# B&R Automation Studio project SampleProject
Automation Studio 4.6.7.161 SP; This is a sample project

## Configuration X20CP1586

CPU X20CP1586, AutomationRuntime B4.63, Build 4.1.2, Vc V4.62.0

### Task classes (Cpu.sw)
```
Cyclic#4:
  Program <- Program.prg
Libraries: AsNxCoM, runtime
```

### Hardware
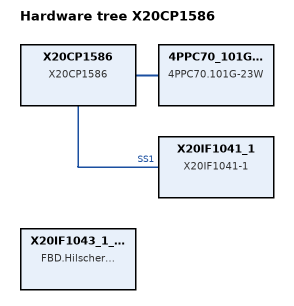
```
4PPC70_101G_23W : 4PPC70.101G-23W v1.4.0.0  [IF2 -> X20CP1586.IF2 [Cable Type=PowerlinkCable, Length=10, Version=1.0.0.2]]
  Connector IF2
  Terminal = true
  KeyMappingFile = VC\4PPC70_101G_23W1.dis
X20CP1586 : X20CP1586 v1.10.0.0
  Connector IF2:
    ActivateDevice = 1
    Mode = Manual
    InternetAddress = 10.0.0.5
    SubnetMask = 255.255.255.0
  ConfigurationID = SampleProject_X20CP1586
X20IF1041_1 : X20IF1041-1 v1.4.0.0  [SS -> X20CP1586.SS1]
  Connector IF1:
    DtmId = 2d840d1b-1473-49bf-a3aa-9ba4bb4caccd
  ConfigFile = X20IF1041_1.dtm
  ConfigModule = asnxdb1
X20IF1043_1__DTM_ : FBD.Hilscher.COGenSlaveDTM.X20IF1043-1 (BuR-X20IF1043-1.eds) v0xA70B.0x00020014 (OrderNumber=X20IF1043-1 (DTM), VendorAddress=2)
  DtmId = 
  ChannelBlocks_722b6533-4489-40d8-aae4-ca0f676f7389  // RxPDO_01
  IO_d52191ed-4c54-4aa1-a555-7a825949a8e7  // 1 Byte(s)
  IO_af2aac78-a722-4896-b9e5-1e0a5520eff8  // 1 Byte(s)
  IO_d3d611f7-76ca-4a12-9739-4a5263261990  // 1 Byte(s)
  IO_28b2f819-6018-4271-9e84-a707596ceac6  // 1 Byte(s)
  IO_602cc8aa-9b3a-44f0-8874-f1db9f83001c  // 1 Byte(s)
  IO_ddc36243-cae0-4301-b86b-f666f3c64e48  // 1 Byte(s)
  IO_1c4766d3-e1da-4921-8d87-31443da98228  // 1 Byte(s)
  IO_b8dce777-eb45-4337-9ffb-03c754224648  // 1 Byte(s)
  ChannelBlocks_8ed83e9a-ae4b-4b45-a0a9-fc1bb8b705e1  // RxPDO_02
  IO_ee120ad1-81d2-4465-b35d-721146a1a332  // 1 Byte(s)
  IO_19650846-5f72-44c2-b9fe-403733023f40  // 1 Byte(s)
  IO_7738ffe0-6403-4fb1-8263-19848970e7e6  // 1 Byte(s)
  IO_6fe8a185-5111-4af8-bbfc-95a7497bd028  // 1 Byte(s)
  IO_049ba4af-e80a-4ae3-8440-0f18dcbcee35  // 1 Byte(s)
  IO_8b1abd60-5eef-4bde-acd4-b9ff9ef701bf  // 1 Byte(s)
  IO_d0747008-f825-4f1e-bb1b-93a7cf56cb81  // 1 Byte(s)
  IO_c2f4c436-f256-4d0e-8b66-210290ce442f  // 1 Byte(s)
  ChannelBlocks_1db14d39-2e65-4f01-bc05-86015beae453  // RxPDO_03
  IO_3ee0241e-3cfb-4054-801c-74f6996894b1  // 1 Byte(s)
  IO_789b20b5-0e27-465d-97d3-aed39c6f7b4d  // 1 Byte(s)
  IO_d9629a54-0cdc-4e26-b1cc-0f655d7bb79f  // 1 Byte(s)
  IO_a93ca36c-91d5-41c1-915d-1e4cef6a746b  // 1 Byte(s)
  IO_44ca810e-2581-480c-9b94-579ce733f4b7  // 1 Byte(s)
  IO_984bf984-2e1d-45ca-ab11-e03385754100  // 1 Byte(s)
  IO_3cd7342f-1a3c-4cf9-8ec7-0170b8e06b47  // 1 Byte(s)
  IO_e044fedb-29b7-41a4-94d1-1d44f9408bcf  // 1 Byte(s)
  ChannelBlocks_33ebcf44-3191-4247-9018-03441b781fe0  // RxPDO_04
  IO_6491ab94-007b-49f2-8672-c682e9e2e849  // 1 Byte(s)
  IO_460835e5-b8fa-402e-a324-cc668286b199  // 1 Byte(s)
  IO_5b7d73de-ee35-47d5-b46d-6039ffd4758c  // 1 Byte(s)
  IO_9b243a73-0c8a-489e-a35b-5add7f9c92f1  // 1 Byte(s)
  IO_2cd10077-e43a-4b7d-9aaf-b023667561cc  // 1 Byte(s)
  IO_0d8de401-27e5-4c9d-967e-d8547063eb60  // 1 Byte(s)
  IO_7a1dea3c-9662-43fd-bbbf-d79c8de14278  // 1 Byte(s)
  IO_cc53336f-8a1e-453e-8010-e83ee473a7c8  // 1 Byte(s)
  ChannelBlocks_469c14d8-50fb-4666-b427-558b6868a6b2  // TxPDO_01
  IO_3dc16d71-7665-442f-942f-20bfc4200c07  // 1 Byte(s)
  IO_9f44e063-2918-4dfd-8b65-24a8848a3e41  // 1 Byte(s)
  IO_3081e22a-489b-4814-96f4-7830738e10a8  // 1 Byte(s)
  IO_468fc6b4-0531-4606-892f-47b44e3cb256  // 1 Byte(s)
  IO_f29869c7-5a2a-4821-8ed8-96205c8678d6  // 1 Byte(s)
  IO_6aec5769-dbad-44db-a853-87637a9343c2  // 1 Byte(s)
  IO_588c8cb2-3609-4ef7-b502-7e643bdfafaa  // 1 Byte(s)
  IO_28ac2c12-4e5d-4a70-9ec7-ebcda2b29e65  // 1 Byte(s)
  ChannelBlocks_ff888c7d-f943-45e3-86a6-88626addf11a  // TxPDO_02
  IO_b3b63fcd-fb3e-44af-8e22-a2afbd636279  // 1 Byte(s)
  IO_a004cc3d-b731-4e23-9db0-44f9f61ab8c5  // 1 Byte(s)
  IO_878c8a23-3a63-42e1-94e4-b06cf4c9534d  // 1 Byte(s)
  IO_e1b211e9-3a5b-4a2e-a15e-f5739b165c14  // 1 Byte(s)
  IO_a27cc85b-b89c-42db-a256-cc393843b87f  // 1 Byte(s)
  IO_c7a2e306-c20a-422f-8e7f-1100758b050e  // 1 Byte(s)
  IO_e2b7146d-279b-4576-961f-e4dc44c5cc91  // 1 Byte(s)
  IO_32390b54-27be-4969-a962-be4e61a52291  // 1 Byte(s)
  ChannelBlocks_05f44e41-c9ab-4a47-be64-14681b8f9c9a  // TxPDO_03
  IO_89de0217-4551-41d6-bedf-6fc1037f9145  // 1 Byte(s)
  IO_8558e8d0-b71d-4751-b843-e24e0b3fc0b9  // 1 Byte(s)
  IO_f8f21e21-716b-4d5c-9128-bc0bbb765fee  // 1 Byte(s)
  IO_1f83f021-3c42-4f7a-972c-2e5081dfceaa  // 1 Byte(s)
  IO_14451fa2-10f8-4e29-8518-78d22b090c99  // 1 Byte(s)
  IO_552231b1-7c23-492d-8bcb-70ee2c2f9c2f  // 1 Byte(s)
  IO_e81a7161-5d17-49ef-aad6-4bb5bdbdcade  // 1 Byte(s)
  IO_b08a2d20-679b-431e-ac8b-f9c1c285acdf  // 1 Byte(s)
  ChannelBlocks_735eb4df-f689-4a63-a199-47a305cb8457  // TxPDO_04
  IO_d2ce0284-5ba9-41fe-b49f-242c2f72ccfc  // 1 Byte(s)
  IO_1d3dc794-09bd-4475-a419-c266234c6ef9  // 1 Byte(s)
  IO_4b8ca6d3-f498-443a-8b72-8bfd9608de3e  // 1 Byte(s)
  IO_a8a31036-494c-4f0e-9e7f-3352be33aaa3  // 1 Byte(s)
  IO_f9151f47-e501-4668-99aa-8f99583e1065  // 1 Byte(s)
  IO_91b97db1-10eb-4fef-bb01-9941d65ccf42  // 1 Byte(s)
  IO_5b890538-7741-4743-86b3-35a3d31369c4  // 1 Byte(s)
  IO_8494ea38-7ce6-4f7d-bc6d-5e7a2a22c0ed  // 1 Byte(s)
```

## Logical view

Binary libraries used (declarations not repeated): operator, runtime, astime, AsIecCon, AsNxCoM


### Program Logical/Program (IEC)

#### Main.st - Init, cyclic, exit code
```iecst
PROGRAM _INIT
	(* Insert code here *)
	NAME := 'SS1.IF1';
	nxcomStartStop_0(enable := TRUE , pDevice := ADR(NAME) , mode := 1 );
END_PROGRAM

PROGRAM _CYCLIC
	(* Insert code here *)

END_PROGRAM

PROGRAM _EXIT
	(* Insert code here *)

END_PROGRAM
```

#### Variables.var - Local variables
```iecst
VAR
	nxcomStartStop_0 : nxcomStartStop;
	NAME : STRING[80];
END_VAR
```

### Program Logical/LibAsCanOpen2_ST/CAN_L2 (IEC) - for PDOs and Can Layer 2 functions

#### CAN_L2.st - Implementation code
```iecst
(********************************************************************
 * COPYRIGHT -- Bernecker + Rainer
 ********************************************************************
 * Program: CAN_L2
 * File: CAN_L2.st
 * Author: Bernecker + Rainer
 * Created: March 30, 2009
 ********************************************************************
 * Implementation of program CAN_L2
 ********************************************************************)

PROGRAM _INIT

(* General assignments *)
CAN_L2.device:= 'SS1.IF2';  (* determine Interface *)

END_PROGRAM

PROGRAM _CYCLIC

CASE CAN_L2.step OF

	0: (* Register COB ID for reading *)

		CAN_L2.CANopenRegisterCOBID_0.enable:= 1;
		CAN_L2.CANopenRegisterCOBID_0.pDevice:= ADR(CAN_L2.device);
		CAN_L2.CANopenRegisterCOBID_0.cobid:= 16#182;
		CAN_L2.CANopenRegisterCOBID_0.inscribe:= TRUE;
		CAN_L2.CANopenRegisterCOBID_0;  (* Call function block *)
		IF CAN_L2.CANopenRegisterCOBID_0.status = ERR_OK THEN  (* OK *)
			CAN_L2.step:= 1; (* next step *)
		ELSIF CAN_L2.CANopenRegisterCOBID_0.status = ERR_FUB_BUSY THEN (* FBK not yet finished *)
			(* busy *)
		ELSE  (* Error step *)
			CAN_L2.step:= 10;
		END_IF

	1: (* Register COB ID for writing *)

		CAN_L2.CANopenRegisterCOBID_1.enable:= 1;
		CAN_L2.CANopenRegisterCOBID_1.pDevice:= ADR(CAN_L2.device);
		CAN_L2.CANopenRegisterCOBID_1.cobid:= 16#202;
		CAN_L2.CANopenRegisterCOBID_1.inscribe:= TRUE;
		CAN_L2.CANopenRegisterCOBID_1;  (* Call function block *)
		IF CAN_L2.CANopenRegisterCOBID_1.status = ERR_OK THEN  (* OK *)
			CAN_L2.step:= 2; (* next step *)
		ELSIF CAN_L2.CANopenRegisterCOBID_1.status = ERR_FUB_BUSY THEN (* FBK not yet finished *)
			(* busy *)
		ELSE  (* Error step *)
			CAN_L2.step:= 10;
		END_IF

	2:  (*Send NMT "Start remote nodes" *)

		CAN_L2.CANopenNMT_0.enable:= 1;
		CAN_L2.CANopenNMT_0.pDevice:= ADR(CAN_L2.device);
		CAN_L2.CANopenNMT_0.node:= 2;  (* node ID 2 *)
		CAN_L2.CANopenNMT_0.state:= coSTART_REMOTE_NODE;  (* Command start remote node *)
		CAN_L2.CANopenNMT_0;  (* Call function block *)
		IF CAN_L2.CANopenNMT_0.status = ERR_OK THEN  (* OK *)
			CAN_L2.step:= 3; (* next step *)
		ELSIF CAN_L2.CANopenNMT_0.status = ERR_FUB_BUSY THEN (* FBK not yet finished *)
			(* busy *)
		ELSE  (* Error step *)
			CAN_L2.step:= 10;
		END_IF

	3: (* Read TPDO1 from IO node *)

		CAN_L2.CANopenPDORead8_0.enable:= 1;
		CAN_L2.CANopenPDORead8_0.pDevice:= ADR(CAN_L2.device);
		CAN_L2.CANopenPDORead8_0.cobid:= 16#182;  (* TPDO1 COB ID *)
		CAN_L2.CANopenPDORead8_0;  (* Call function block *)
		IF CAN_L2.CANopenPDORead8_0.status = ERR_OK THEN  (* OK *)
			CAN_L2.step:= 4; (* next step *)
		ELSIF CAN_L2.CANopenPDORead8_0.status = ERR_FUB_BUSY THEN (* FBK not yet finished *)
			(* busy *)
		ELSE  (* Error step *)
			CAN_L2.step:= 10;
		END_IF

	4: (* Write RPDO1 to IO node *)

		CAN_L2.CANopenPDOWrite8_0.enable:= 1;
		CAN_L2.CANopenPDOWrite8_0.pDevice:= ADR(CAN_L2.device);
		CAN_L2.CANopenPDOWrite8_0.cobid:= 16#202;  (* RPDO1 COB ID *)
		CAN_L2.CANopenPDOWrite8_0.data0:= CAN_L2.Data[0];  (* Data written to the IO device *)
		CAN_L2.CANopenPDOWrite8_0.datalen:= 8;  (* Length of PDO *)
		CAN_L2.CANopenPDOWrite8_0;  (* Call function block *)
		IF CAN_L2.CANopenPDOWrite8_0.status = ERR_OK THEN  (* OK *)
			CAN_L2.Data[0]:= CAN_L2.Data[0] + 1;  (* running counter *)
			CAN_L2.step:= 3; (* next step *)
		ELSIF CAN_L2.CANopenPDOWrite8_0.status = ERR_FUB_BUSY THEN (* FBK not yet finished *)
			(* busy *)
		ELSE  (* Error step *)
			CAN_L2.step:= 10;
		END_IF
END_CASE

END_PROGRAM
```

#### CAN_L2.typ - Local data types
```iecst
(********************************************************************
 * COPYRIGHT -- Bernecker + Rainer
 ********************************************************************
 * Program: CAN_L2
 * File: CAN_L2.typ
 * Author: Bernecker + Rainer
 * Created: March 30, 2009
 ********************************************************************
 * Local data types of program CAN_L2
 ********************************************************************)

TYPE
	CAN_L2_typ : 	STRUCT
		step : USINT;
		device : STRING[80];
		Data : ARRAY[0..7] OF USINT;
		CANopenRegisterCOBID_0 : CANopenRegisterCOBID;
		CANopenRegisterCOBID_1 : CANopenRegisterCOBID;
		CANopenPDORead8_0 : CANopenPDORead8;
		CANopenPDOWrite8_0 : CANopenPDOWrite8;
		CANopenNMT_0 : CANopenNMT;
	END_STRUCT;
END_TYPE
```

#### CAN_L2.var - Local variables
```iecst
(********************************************************************
 * COPYRIGHT -- Bernecker + Rainer
 ********************************************************************
 * Program: CAN_L2
 * File: CAN_L2.var
 * Author: Bernecker + Rainer
 * Created: March 30, 2009
 ********************************************************************
 * Local variables of program CAN_L2
 ********************************************************************)
VAR
	CAN_L2 : CAN_L2_typ := (0);
END_VAR
```

### Program Logical/LibAsCanOpen3_ST/SDO (IEC) - SDO access

#### SDO.st - Implementation code
```iecst
(********************************************************************
 * COPYRIGHT -- Bernecker + Rainer
 ********************************************************************
 * Program: SDO
 * File: SDO.st
 * Author: Bernecker + Rainer
 * Created: March 30, 2009
 ********************************************************************
 * Implementation of program SDO
 ********************************************************************)

PROGRAM _INIT

(* General assignments *)
SDO.device:= 'SS1.IF2';  (* determine Interface *)

END_PROGRAM

PROGRAM _CYCLIC

CASE SDO.step OF

	0: (* Read Device ID form IO node *)

		SDO.CANopenSDORead8_0.enable:= 1;
		SDO.CANopenSDORead8_0.pDevice:= ADR(SDO.device);
		SDO.CANopenSDORead8_0.node:= 2;  (* Node ID from IO device *)
		SDO.CANopenSDORead8_0.index:= 16#100A;  (* Index of IO device; BC0043 = Firmware version *)
		SDO.CANopenSDORead8_0.subindex:= 16#0000; (* Subindex of IO device *)
		SDO.CANopenSDORead8_0;  (* Call function block *)
		IF SDO.CANopenSDORead8_0.status = ERR_OK THEN  (* OK *)
			SDO.step:= 1; (* next step *)
		ELSIF SDO.CANopenSDORead8_0.status = ERR_FUB_BUSY THEN (* FBK not yet finished *)
			(* busy *)
		ELSE  (* Error step *)
			SDO.step:= 10;
		END_IF

	1: (* Configuration of AT6402 card on slot 2 *)
		(* Write Module ID to BC0043 *)

		SDO.CANopenSDOWrite8_0.enable:= 1;
		SDO.CANopenSDOWrite8_0.pDevice:= ADR(SDO.device);
		SDO.CANopenSDOWrite8_0.node:= 2;  (* Node ID from IO device *)
		SDO.CANopenSDOWrite8_0.index:= 16#2251;  (* Index of IO device; BC0043 = Parameter modul 2 *)
		SDO.CANopenSDOWrite8_0.subindex:= 16#01;  (* Subindex of IO device; BC0043 = Get configured module ID *)
		SDO.CANopenSDOWrite8_0.data0:= 16#A9;  (* low byte of module ID *)
		SDO.CANopenSDOWrite8_0.data1:= 16#1B;  (* high byte of module ID *)
		SDO.CANopenSDOWrite8_0.datalen:= 2;
		SDO.CANopenSDOWrite8_0;
		IF SDO.CANopenSDOWrite8_0.status = ERR_OK THEN  (* OK *)
			SDO.step:= 2; (* next step *)
		ELSIF SDO.CANopenSDOWrite8_0.status = ERR_FUB_BUSY THEN (* FBK not yet finished *)
			(* busy *)
		ELSE  (* Error step *)
			SDO.step:= 10;
		END_IF

	2: (* Configuration of AT6402 card on slot 2 *)
		(* Write Sensor Type J to AT6402 *)

		SDO.CANopenSDOWrite8_1.enable:= 1;
		SDO.CANopenSDOWrite8_1.pDevice:= ADR(SDO.device);
		SDO.CANopenSDOWrite8_1.node:= 2;  (* Node ID from IO device *)
		SDO.CANopenSDOWrite8_1.index:= 16#2251;  (* Index of IO device; BC0043 = Parameter modul 2 *)
		SDO.CANopenSDOWrite8_1.subindex:= 16#0A;  (* Subindex of IO device; BC0043 = Parameter 1 modul 2*)
		SDO.CANopenSDOWrite8_1.data0:= 16#02;  (* low byte of config data *)
		SDO.CANopenSDOWrite8_1.data1:= 16#00;  (* high byte of config data *)
		SDO.CANopenSDOWrite8_1.data2:= 16#1A;  (* low byte of register number *)
		SDO.CANopenSDOWrite8_1.data3:= 16#00;  (* high byte of register number *)
		SDO.CANopenSDOWrite8_1.datalen:= 4;
		SDO.CANopenSDOWrite8_1;
		IF SDO.CANopenSDOWrite8_1.status = ERR_OK THEN  (* OK *)
			SDO.step:= 3; (* next step *)
		ELSIF SDO.CANopenSDOWrite8_1.status = ERR_FUB_BUSY THEN (* FBK not yet finished *)
			(* busy *)
		ELSE  (* Error step *)
			SDO.step:= 10;
		END_IF

	3: (* Configuration of AT6402 card on slot 2 *)
		(* Disable input 2-6 *)

		SDO.CANopenSDOWrite8_2.enable:= 1;
		SDO.CANopenSDOWrite8_2.pDevice:= ADR(SDO.device);
		SDO.CANopenSDOWrite8_2.node:= 2;  (* Node ID from IO device *)
		SDO.CANopenSDOWrite8_2.index:= 16#2251;  (* Index of IO device; BC0043 = Parameter modul 2*)
		SDO.CANopenSDOWrite8_2.subindex:= 16#0B;  (* Subindex of IO device; BC0043 = Parameter 2 modul 2 *)
		SDO.CANopenSDOWrite8_2.data0:= 16#01;  (* low byte of config data *)
		SDO.CANopenSDOWrite8_2.data1:= 16#00;  (* high byte of config data *)
		SDO.CANopenSDOWrite8_2.data2:= 16#1B;  (* low byte of register number *)
		SDO.CANopenSDOWrite8_2.data3:= 16#00;  (* high byte of register number *)
		SDO.CANopenSDOWrite8_2.datalen:= 4;
		SDO.CANopenSDOWrite8_2;
		IF SDO.CANopenSDOWrite8_2.status = ERR_OK THEN  (* OK *)
			SDO.step:= 4; (* next step *)
		ELSIF SDO.CANopenSDOWrite8_2.status = ERR_FUB_BUSY THEN (* FBK not yet finished *)
			(* busy *)
		ELSE  (* Error step *)
			SDO.step:= 10;
		END_IF

	4: (* Configuration of AT6402 card on slot 2 *)
		(* Store configuration on BC0043 *)

		SDO.CANopenSDOWrite8_3.enable:= 1;
		SDO.CANopenSDOWrite8_3.pDevice:= ADR(SDO.device);
		SDO.CANopenSDOWrite8_3.node:= 2;  (* Node ID from IO device *)
		SDO.CANopenSDOWrite8_3.index:= 16#1010;  (* Index of IO device; BC0043 = Store parameter field *)
		SDO.CANopenSDOWrite8_3.subindex:= 16#01;  (* Subindex of IO device; BC0043 = save all parameter *)
		SDO.CANopenSDOWrite8_3.data0:= 16#73;  (* low byte of config data *)
		SDO.CANopenSDOWrite8_3.data1:= 16#61;  (* high byte of config data *)
		SDO.CANopenSDOWrite8_3.data2:= 16#76;  (* low byte of register number *)
		SDO.CANopenSDOWrite8_3.data3:= 16#65;  (* high byte of register number *)
		SDO.CANopenSDOWrite8_3.datalen:= 4;
		SDO.CANopenSDOWrite8_3;
		IF SDO.CANopenSDOWrite8_3.status = ERR_OK THEN  (* OK *)
			SDO.step:= 5; (* next step *)
		ELSIF SDO.CANopenSDOWrite8_3.status = ERR_FUB_BUSY THEN (* FBK not yet finished *)
			(* busy *)
		ELSE  (* Error step *)
			SDO.step:= 10;
		END_IF

END_CASE

END_PROGRAM
```

#### SDO.typ - Local data types
```iecst
(********************************************************************
 * COPYRIGHT -- Bernecker + Rainer
 ********************************************************************
 * Program: SDO
 * File: SDO.typ
 * Author: Bernecker + Rainer
 * Created: March 30, 2009
 ********************************************************************
 * Local data types of program SDO
 ********************************************************************)

TYPE
	SDO_type : 	STRUCT
		step : USINT;
		device : STRING[80];
		CANopenSDORead8_0 : CANopenSDORead8;
		CANopenSDOWrite8_0 : CANopenSDOWrite8;
		CANopenSDOWrite8_1 : CANopenSDOWrite8;
		CANopenSDOWrite8_2 : CANopenSDOWrite8;
		CANopenSDOWrite8_3 : CANopenSDOWrite8;
	END_STRUCT;
END_TYPE
```

#### SDO.var - Local variables
```iecst
(********************************************************************
 * COPYRIGHT -- Bernecker + Rainer
 ********************************************************************
 * Program: SDO
 * File: SDO.var
 * Author: Bernecker + Rainer
 * Created: March 30, 2009
 ********************************************************************
 * Local variables of program SDO
 ********************************************************************)
VAR
	SDO : SDO_type := (0);
END_VAR
```

Listed in the project but not available here: Logical/Global.typ, Logical/Global.var, Logical/Program/Types.typ
